FUNCTION_BLOCK IED50 (* Extracted Composite Function Block Type *)
  (* Version 3/29/2017, bdowdesw *)
  PACKAGE Main;
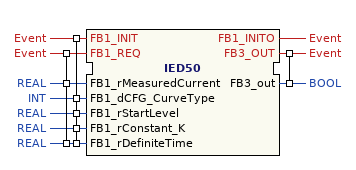
  EVENT_INPUT
    FB1_INIT WITH FB1_dCFG_CurveType, FB1_rStartLevel, FB1_rConstant_K, FB1_rDefiniteTime; (* Initialization Request *)
    FB1_REQ WITH FB1_rMeasuredCurrent, FB1_rDefiniteTime; (* Normal Execution Request *)
  END_EVENT
  EVENT_OUTPUT
    FB1_INITO; (* Initialization Confirm *)
    FB3_OUT WITH FB3_out; (* Execution Confirmation *)
  END_EVENT
  VAR_INPUT
    FB1_rMeasuredCurrent : REAL; (* Input event qualifier *)
    FB1_dCFG_CurveType : INT;
    FB1_rStartLevel : REAL;
    FB1_rConstant_K : REAL;
    FB1_rDefiniteTime : REAL;
  END_VAR
  VAR_OUTPUT
    FB3_out : BOOL; (* Output event qualifier *)
  END_VAR
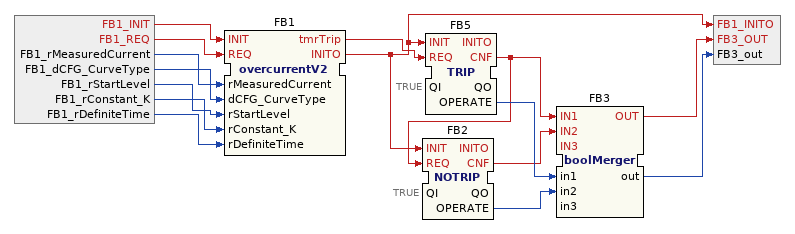
  FBS
    FB5 : TRIP(QI := TRUE);
    FB1 : overcurrentV2;
    FB2 : NOTRIP(QI := TRUE);
    FB3 : boolMerger;
  END_FBS
  EVENT_CONNECTIONS
    FB1.tmrTrip TO FB5.REQ;
    FB1.INITO TO FB5.INIT;
    FB5.CNF TO FB3.IN1;
    FB2.CNF TO FB3.IN2;
    FB1.INITO TO FB2.INIT;
    FB5.CNF TO FB2.REQ;
    FB1_INIT TO FB1.INIT;
    FB1_REQ TO FB1.REQ;
    FB1.INITO TO FB1_INITO;
    FB3.OUT TO FB3_OUT;
  END_CONNECTIONS
  DATA_CONNECTIONS
    FB5.OPERATE TO FB3.in1;
    FB2.OPERATE TO FB3.in2;
    FB1_rMeasuredCurrent TO FB1.rMeasuredCurrent;
    FB1_dCFG_CurveType TO FB1.dCFG_CurveType;
    FB1_rStartLevel TO FB1.rStartLevel;
    FB1_rConstant_K TO FB1.rConstant_K;
    FB1_rDefiniteTime TO FB1.rDefiniteTime;
    FB3.out TO FB3_out;
  END_CONNECTIONS
END_FUNCTION_BLOCK
